(*

## Short summary

This class provides assert statements for date and time types with 32 bit length
It implements the interface `ISimpleDateAndTimeAssertions`
For date and time (``DT``) use `SimpleDateAndTimeAssertions.dateAndTime`
For date (``DATE``) use  `SimpleDateAndTimeAssertions.dateOnly`
For time of day (``TOD``) use  `SimpleDateAndTimeAssertions.timeOfDay`

.. <legal notes>

legal notes
=================
| SPDX-FileCopyrightText: © 2022 ekvip automation GmbH <info@ekvip.de>
| SPDX-License-Identifier: Apache-2.0
| For details check: Apache-2.0_

.. _Apache-2.0: https://www.apache.org/licenses/LICENSE-2.0

.. </legal notes>



*)

{attribute 'reflection'}
FUNCTION_BLOCK INTERNAL LongDateAndTimeAssertions 
EXTENDS CNM_AbstractObject.Object
IMPLEMENTS ILongDateAndTimeAssertions, IAssertCallBacksetter
VAR
	(* class to handle date assertions *)
	dateAssertions		:DateAssertions64Bit();
	(* class to handle date and time assertions *)
	dateTimeAssertions	:DateTimeAssertions64Bit();
	(* class to handle time of day assertions *)
	timeOfDayAssertions	:TimeOfDayAssertions64Bit();
END_VAR

(*

## Short summary
This abstract property returns the class name of the concrete object, 
It's for debugging purpose

.. <legal notes>

legal notes
=================
| SPDX-FileCopyrightText: © 2022 ekvip automation GmbH <info@ekvip.de>
| SPDX-License-Identifier: Apache-2.0
| For details check: Apache-2.0_

.. _Apache-2.0: https://www.apache.org/licenses/LICENSE-2.0

.. </legal notes>

*)

PROPERTY className :CNM_AbstractObject.ClassName
GET
className := 'CNM_Assertor.LongDateAndTimeAssertions';
END_GET
END_PROPERTY

(*

## Short summary
Returns the interface `I32BitDtAssertions`
with assert statements for 32 bit date and time ``DT``

.. <legal notes>

legal notes
=================
| SPDX-FileCopyrightText: © 2022 ekvip automation GmbH <info@ekvip.de>
| SPDX-License-Identifier: Apache-2.0
| For details check: Apache-2.0_

.. _Apache-2.0: https://www.apache.org/licenses/LICENSE-2.0

.. </legal notes>

*)

PROPERTY dateAndTime :I64BitDtAssertions
GET
dateAndTime := THIS^.dateTimeAssertions;
END_GET
END_PROPERTY

(*

## Short summary
Returns the interface `I32BitDateAssertions`
with assert statements for 32 bit date ``DATE``

.. <legal notes>

legal notes
=================
| SPDX-FileCopyrightText: © 2022 ekvip automation GmbH <info@ekvip.de>
| SPDX-License-Identifier: Apache-2.0
| For details check: Apache-2.0_

.. _Apache-2.0: https://www.apache.org/licenses/LICENSE-2.0

.. </legal notes>

*)

PROPERTY dateOnly : I64BitDateAssertions
GET
dateOnly := THIS^.dateAssertions;
END_GET
END_PROPERTY

(*

## Short summary
This methods is the setter for the callback class if an assertion was false

.. <legal notes>

legal notes
=================
| SPDX-FileCopyrightText: © 2022 ekvip automation GmbH <info@ekvip.de>
| SPDX-License-Identifier: Apache-2.0
| For details check: Apache-2.0_

.. _Apache-2.0: https://www.apache.org/licenses/LICENSE-2.0

.. </legal notes>



*)

METHOD setCallBack
VAR_INPUT
	(* the class that must be informed if an assertion is false *)
	callBack	:IAssertCallBack;  
END_VAR
THIS^.dateAssertions.setCallBack(callBack);
THIS^.dateTimeAssertions.setCallBack(callBack);
THIS^.timeOfDayAssertions.setCallBack(callBack);
END_METHOD

(*

## Short summary
Returns the interface `I32BitDateAssertions`
with assert statements for 32 bit time of day ``TOD``

.. <legal notes>

legal notes
=================
| SPDX-FileCopyrightText: © 2022 ekvip automation GmbH <info@ekvip.de>
| SPDX-License-Identifier: Apache-2.0
| For details check: Apache-2.0_

.. _Apache-2.0: https://www.apache.org/licenses/LICENSE-2.0

.. </legal notes>

*)

PROPERTY timeOfDay :I64BitTodAssertions
GET
timeOfDay := THIS^.timeOfDayAssertions;
END_GET
END_PROPERTY

END_FUNCTION_BLOCK

(* stored: Version 1.1.0.1, ProductVersion 3.1.4026.12
   POU LongDateAndTimeAssertions: Id {947be7dd-b3de-461b-b26a-dd355d77593e}, SpecialFunc None
   Property className: Id {eadd6b85-18f9-4ae5-ad0d-6130e594c18b}
   Get Get: Id {b8a6da0c-248f-41dc-8539-2cbd15766e5a}
   Property dateAndTime: Id {ce6f37b5-d21f-4bae-a6d4-ca1d6990b4b6}
   Get Get: Id {56d2f47a-ae00-41d0-8bd0-5e793583e342}
   Property dateOnly: Id {b23fb871-cc6a-4d6d-89c0-c4d86f0c2b0f}
   Get Get: Id {3ccc87a8-7e8d-44b7-b100-a889ec8ac476}
   Method setCallBack: Id {4b8d3625-1b81-4e9d-b616-1d479fbbf21e}
   Property timeOfDay: Id {ca33e8ed-d3e3-473f-9231-ec1a8ded05fc}
   Get Get: Id {e4b7b3b2-041d-484e-87dd-ab66474e22ea} *)
